INTERFACE ITF_Cylinder

PROPERTY Extended : BOOL
GET
END_GET
END_PROPERTY

METHOD METH_Extend : BOOL
END_METHOD

METHOD METH_Retract : BOOL
END_METHOD

PROPERTY Retracted : BOOL
GET
END_GET
END_PROPERTY

END_INTERFACE

(* stored: Version 1.1.0.1
   Itf ITF_Cylinder: Id {b5cb89fb-8b89-4247-8945-39522e8706bd}
   Property Extended: Id {09fb00ae-d1fc-42c0-ad57-6aa0b0b0b39f}
   Get Get: Id {2dd3f90c-9c72-4543-9a31-ce04c185a95f}
   Method METH_Extend: Id {042e18f7-e957-4643-96ae-afb65fe40d6c}
   Method METH_Retract: Id {1495efb4-865b-4797-a4fb-33004ed07a7c}
   Property Retracted: Id {af487719-1e3f-4066-9881-1016aed0ce28}
   Get Get: Id {367af784-97e0-4f04-93a8-c59f01a01e06} *)
